TYPE "PLCtoMES_MainCheckOutStation2ST350_ext"
VERSION : 0.1
   STRUCT
      CheckSum : Int;
      PartTypeID : Int;
      PartTypeSN : String[60];
      PalletID : Int;
      PartStatus : Int;
      SubPartSN : String[60];
      "Transfer time" : String[60];
      Spare : Array[194..998] of Byte;
      Massage { S7_SetPoint := 'False'} : "PLCtoMES_AlarmMassage_ext";
   END_STRUCT;

END_TYPE

